TYPE GreenMasterParametersXXL:
STRUCT
	System: SystemParametersXXL;
END_STRUCT
END_TYPE

(* stored: Version 1.1.0.1, ProductVersion 3.1.4024.6
   DUT GreenMasterParametersXXL: Id {b1e94a17-75ad-4bc1-864b-01c5f39120d1} *)
